SUBAPPLICATION Knickdeichsel (* Subapplication Type *)
  (* Standard: 61499-2 *)
  (* Version 1.0, 2023-01-29, Franz *)
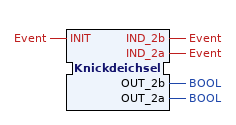
  EVENT_INPUT
    INIT;
  END_EVENT
  EVENT_OUTPUT
    IND_2b;
    IND_2a;
  END_EVENT
  VAR_OUTPUT
    OUT_2b : BOOL;
    OUT_2a : BOOL;
  END_VAR
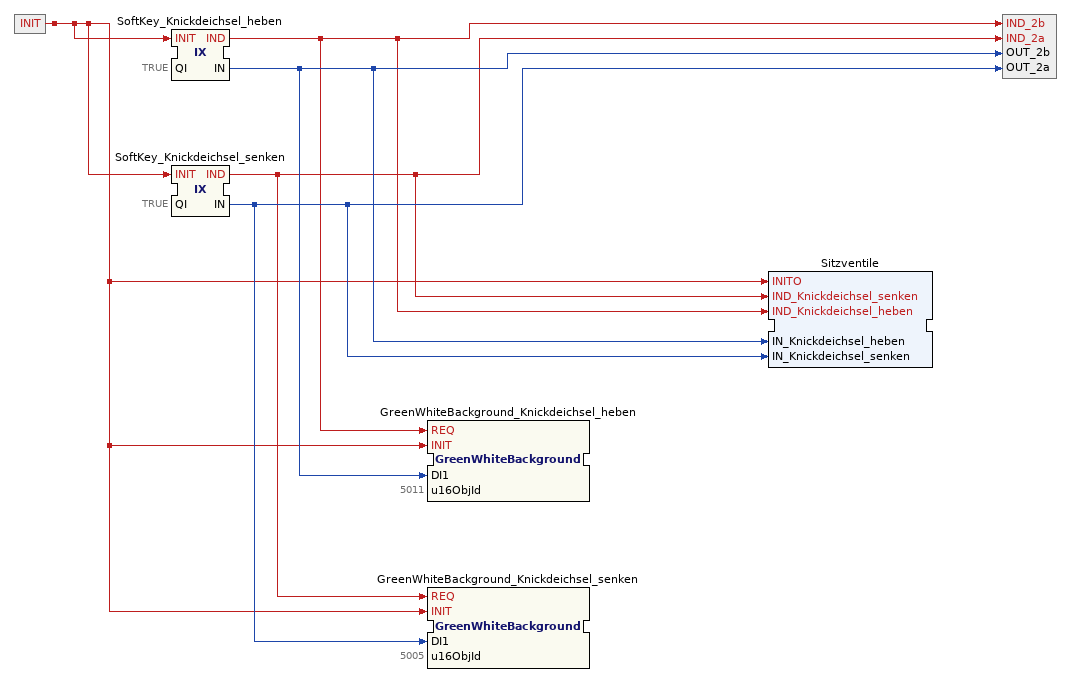
  FBS
    SoftKey_Knickdeichsel_heben : IX(QI := TRUE);
    SoftKey_Knickdeichsel_senken : IX(QI := TRUE);
    GreenWhiteBackground_Knickdeichsel_senken : GreenWhiteBackground(u16ObjId := 5005);
    GreenWhiteBackground_Knickdeichsel_heben : GreenWhiteBackground(u16ObjId := 5011);
  END_FBS
  SUBAPPLICATION Sitzventile (* Sitzventile *)
    EVENT_INPUT
      INITO;
      IND_Knickdeichsel_senken;
      IND_Knickdeichsel_heben;
    END_EVENT
    VAR_INPUT
      IN_Knickdeichsel_heben : BOOL;
      IN_Knickdeichsel_senken : BOOL;
    END_VAR
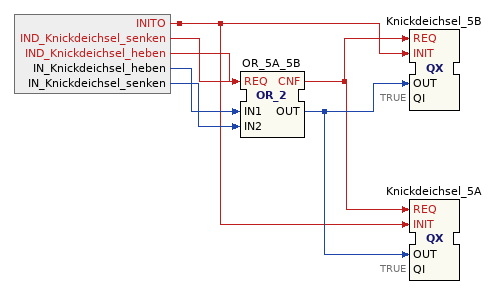
    FBS
      OR_5A_5B : OR_2; {SET_ATTRIBUTE(PinComment, IN1:Knickdeichsel_heben)} {SET_ATTRIBUTE(PinComment, IN2:Knickdeichsel_senken)}
      Knickdeichsel_5B : QX(QI := TRUE);
      Knickdeichsel_5A : QX(QI := TRUE);
    END_FBS
    EVENT_CONNECTIONS
      OR_5A_5B.CNF TO Knickdeichsel_5B.REQ;
      OR_5A_5B.CNF TO Knickdeichsel_5A.REQ;
      IND_Knickdeichsel_senken TO OR_5A_5B.REQ;
      IND_Knickdeichsel_heben TO OR_5A_5B.REQ;
      INITO TO Knickdeichsel_5B.INIT;
      INITO TO Knickdeichsel_5A.INIT;
    END_CONNECTIONS
    DATA_CONNECTIONS
      OR_5A_5B.OUT TO Knickdeichsel_5B.OUT;
      OR_5A_5B.OUT TO Knickdeichsel_5A.OUT;
      IN_Knickdeichsel_heben TO OR_5A_5B.IN1;
      IN_Knickdeichsel_senken TO OR_5A_5B.IN2;
    END_CONNECTIONS
  END_SUBAPPLICATION
  EVENT_CONNECTIONS
    SoftKey_Knickdeichsel_heben.IND TO GreenWhiteBackground_Knickdeichsel_heben.REQ;
    SoftKey_Knickdeichsel_senken.IND TO GreenWhiteBackground_Knickdeichsel_senken.REQ;
    INIT TO SoftKey_Knickdeichsel_heben.INIT;
    SoftKey_Knickdeichsel_heben.IND TO IND_2b;
    INIT TO SoftKey_Knickdeichsel_senken.INIT;
    SoftKey_Knickdeichsel_senken.IND TO IND_2a;
    SoftKey_Knickdeichsel_senken.IND TO Sitzventile.IND_Knickdeichsel_senken;
    SoftKey_Knickdeichsel_heben.IND TO Sitzventile.IND_Knickdeichsel_heben;
    INIT TO Sitzventile.INITO;
    INIT TO GreenWhiteBackground_Knickdeichsel_heben.INIT;
    INIT TO GreenWhiteBackground_Knickdeichsel_senken.INIT;
  END_CONNECTIONS
  DATA_CONNECTIONS
    SoftKey_Knickdeichsel_heben.IN TO GreenWhiteBackground_Knickdeichsel_heben.DI1;
    SoftKey_Knickdeichsel_senken.IN TO GreenWhiteBackground_Knickdeichsel_senken.DI1;
    SoftKey_Knickdeichsel_heben.IN TO OUT_2b;
    SoftKey_Knickdeichsel_senken.IN TO OUT_2a;
    SoftKey_Knickdeichsel_heben.IN TO Sitzventile.IN_Knickdeichsel_heben;
    SoftKey_Knickdeichsel_senken.IN TO Sitzventile.IN_Knickdeichsel_senken;
  END_CONNECTIONS
END_SUBAPPLICATION
